{region '#Template'}
	{attribute 'Version' := '1.2.0.0'}
	{attribute 'Tags' := '"LCID": "1031", "Text": "Plant, Weatherstation, Draft"'}
	{attribute 'Tags' := '"LCID": "1033", "Text": "Plant, Weatherstation, Draft"'}
	{attribute 'Description' := '"LCID": "1031", "Text": "Vorlage-Template: beinhaltet alle Objekte, die Eingangsverknüpfung zu diesen muss vom Anwender erstellt werden"'}
	{attribute 'Description' := '"LCID": "1033", "Text": "Draft-template: contains all objects to be connected to appropriate inputs by the user"'}
{endregion}
FUNCTION_BLOCK FB_BA_WeatherStation_Draft EXTENDS FB_BA_View
VAR_INPUT CONSTANT
	Dstb						: FB_BA_SensorBinary;
	Rain						: FB_BA_SensorBinary;
	WthT						: FB_BA_SensorAnalog;
	DewPtT						: FB_BA_SensorAnalog; 
	PrssAbs						: FB_BA_SensorAnalog;
	PrssRel						: FB_BA_SensorAnalog;
	HumAbs						: FB_BA_SensorAnalog;
	HumRel						: FB_BA_SensorAnalog;
	Brightness					: FB_BA_MeasuredValueCardinal;
	Dawn						: FB_BA_SensorAnalog;
	GlobRadn					: FB_BA_SensorAnalog;      
	WndDir						: FB_BA_SensorAnalog;
	WndSpd						: FB_BA_SensorAnalog; 
	Latd						: FB_BA_SensorAnalog;  
	Lngt						: FB_BA_SensorAnalog; 
	SunAzm						: FB_BA_SensorAnalog;
	SunElv						: FB_BA_SensorAnalog;                 
END_VAR	

VAR
	WeatherStation				: FB_BA_RawPublisher;
	stWeatherStation			: ST_BA_WeatherStation;
	stDateTime_PLACEHOLDER		: TIMESTRUCT;			// Placeholder-variable, so the template can be compiled correctly
														// to be replaced by an appropriate timestruct
END_VAR

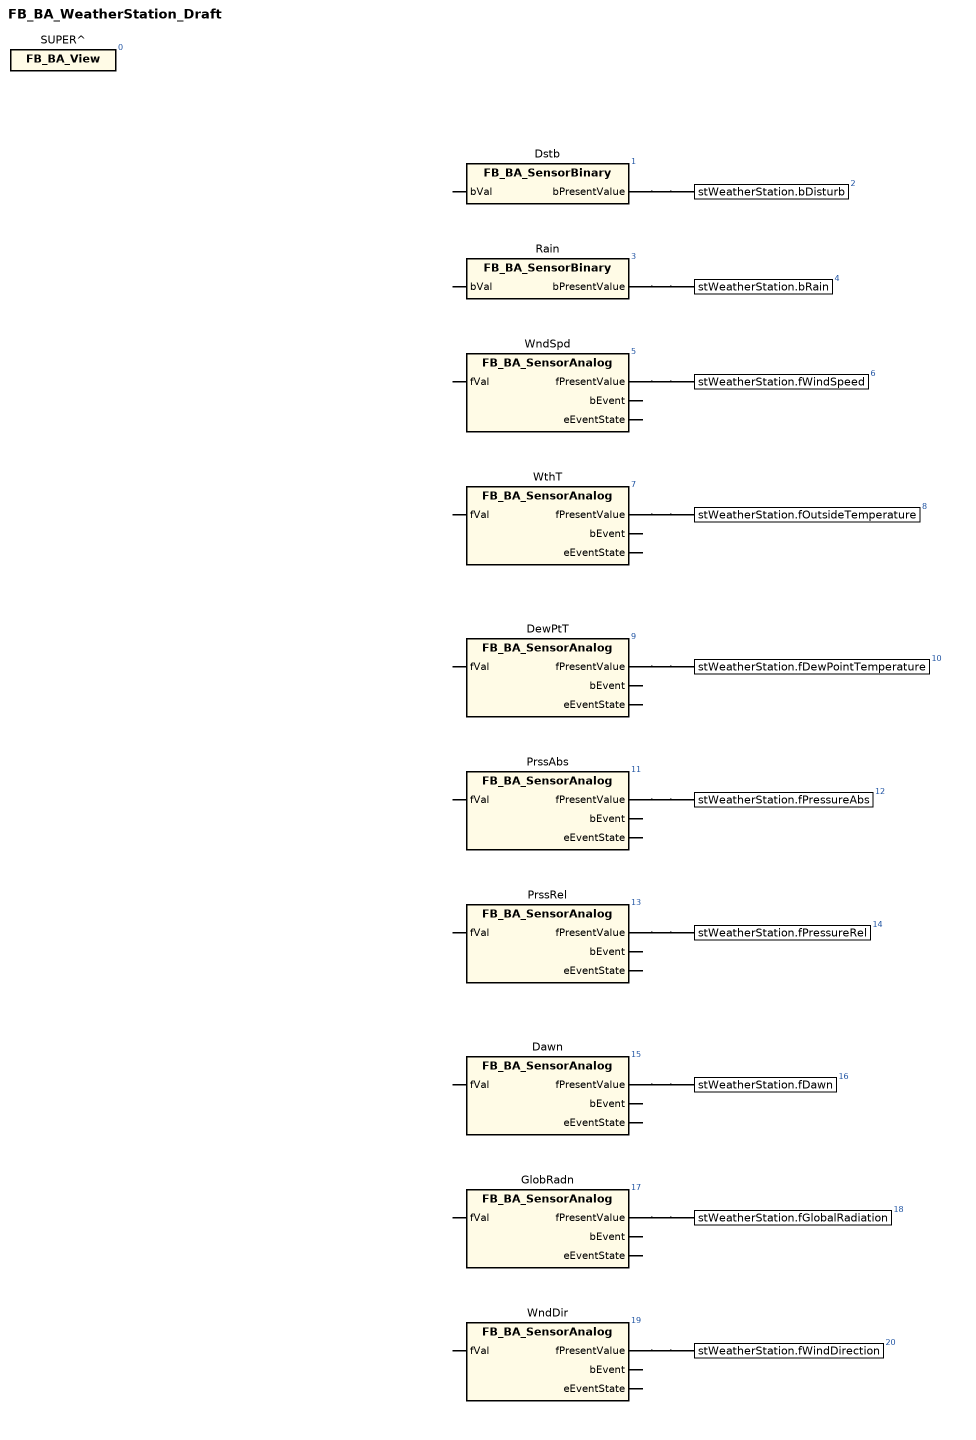
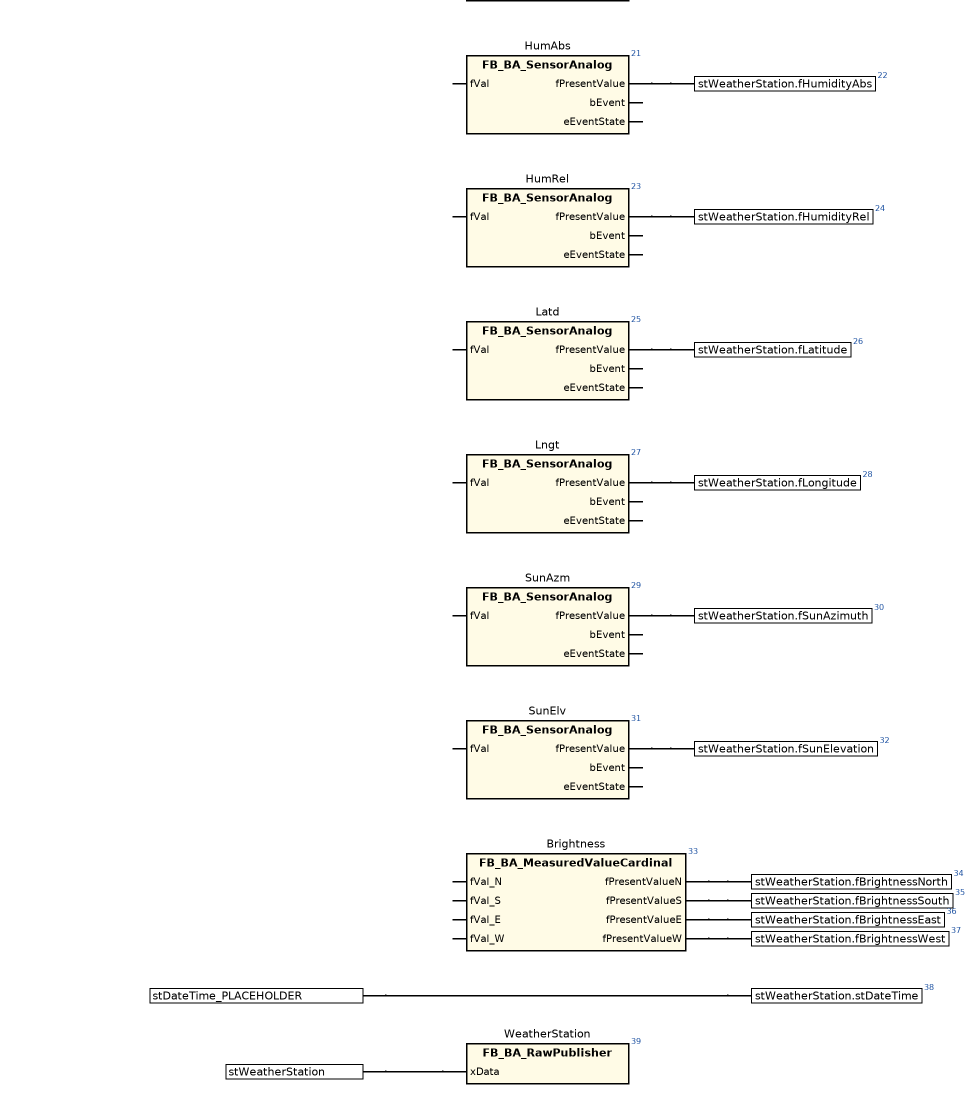
SUPER^(); // FB_BA_View
Dstb(); // FB_BA_SensorBinary
stWeatherStation.bDisturb := Dstb.bPresentValue;
Rain(); // FB_BA_SensorBinary
stWeatherStation.bRain := Rain.bPresentValue;
WndSpd(); // FB_BA_SensorAnalog
stWeatherStation.fWindSpeed := WndSpd.fPresentValue;
WthT(); // FB_BA_SensorAnalog
stWeatherStation.fOutsideTemperature := WthT.fPresentValue;
DewPtT(); // FB_BA_SensorAnalog
stWeatherStation.fDewPointTemperature := DewPtT.fPresentValue;
PrssAbs(); // FB_BA_SensorAnalog
stWeatherStation.fPressureAbs := PrssAbs.fPresentValue;
PrssRel(); // FB_BA_SensorAnalog
stWeatherStation.fPressureRel := PrssRel.fPresentValue;
Dawn(); // FB_BA_SensorAnalog
stWeatherStation.fDawn := Dawn.fPresentValue;
GlobRadn(); // FB_BA_SensorAnalog
stWeatherStation.fGlobalRadiation := GlobRadn.fPresentValue;
WndDir(); // FB_BA_SensorAnalog
stWeatherStation.fWindDirection := WndDir.fPresentValue;
HumAbs(); // FB_BA_SensorAnalog
stWeatherStation.fHumidityAbs := HumAbs.fPresentValue;
HumRel(); // FB_BA_SensorAnalog
stWeatherStation.fHumidityRel := HumRel.fPresentValue;
Latd(); // FB_BA_SensorAnalog
stWeatherStation.fLatitude := Latd.fPresentValue;
Lngt(); // FB_BA_SensorAnalog
stWeatherStation.fLongitude := Lngt.fPresentValue;
SunAzm(); // FB_BA_SensorAnalog
stWeatherStation.fSunAzimuth := SunAzm.fPresentValue;
SunElv(); // FB_BA_SensorAnalog
stWeatherStation.fSunElevation := SunElv.fPresentValue;
Brightness(); // FB_BA_MeasuredValueCardinal
stWeatherStation.fBrightnessNorth := Brightness.fPresentValueN;
stWeatherStation.fBrightnessSouth := Brightness.fPresentValueS;
stWeatherStation.fBrightnessEast := Brightness.fPresentValueE;
stWeatherStation.fBrightnessWest := Brightness.fPresentValueW;
stWeatherStation.stDateTime := stDateTime_PLACEHOLDER;
WeatherStation(xData := stWeatherStation); // FB_BA_RawPublisher

METHOD FB_init : BOOL
VAR_INPUT
	bInitRetains : BOOL; // if TRUE, the retain variables are initialized (warm start / cold start)
	bInCopyCode : BOOL;  // if TRUE, the instance afterwards gets moved into the copy code (online change)
END_VAR
	Dstb.iParent							:= THIS^;
	Dstb.iLabel 							:= LblAggregates_WeatherStation;							
	Dstb.sObjectName						:= '{Idx=01}';
	Dstb.eDPADMode							:= E_BA_DPADMode.eInclude;		
	Dstb.Input.sActiveText 					:= txtEvent_Triggered;       
	Dstb.Input.sInactiveText 				:= txtEvent_Normal;          
	Dstb.Input.nEventClassID				:= EC_ID.NC30;
	Dstb.Input.aEventTransitionText[1]		:= txtEvent_Triggered;       
	Dstb.Input.aEventTransitionText[2]		:= txtEvent_Error;           
	Dstb.Input.aEventTransitionText[3]		:= txtEvent_Normal;          
	Dstb.Input.bEventDetectionEnable		:= TRUE;                     
                        	
	Rain.iParent							:= THIS^;
	Rain.iLabel 							:= LblAggregates_RainSensor;							
	Rain.sObjectName						:= '{Idx=01}';
	Rain.eDPADMode							:= E_BA_DPADMode.eInclude;		
	Rain.Input.iLabel	 					:= LblFunctions_Status;
	Rain.Input.sActiveText 					:= txtEvent_Yes;
	Rain.Input.sInactiveText 				:= txtEvent_No;
	Rain.Input.nEventClassID				:= EC_ID.NC60;
	Rain.Input.aEventTransitionText[1]		:= txtEvent_No;
	Rain.Input.aEventTransitionText[2]		:= txtEvent_None;
	Rain.Input.aEventTransitionText[3]		:= txtEvent_Yes;
	Rain.Input.bEventDetectionEnable		:= FALSE;	
                        	
	WthT.iParent							:= THIS^;
	WthT.iLabel 							:= LblAggregates_TemperatureOutside;
	WthT.sObjectName						:= '{Idx=01}';
	WthT.eDPADMode							:= E_BA_DPADMode.eInclude;
	WthT.MV.eUnit 							:= E_BA_Unit.eTemperature_DegreesCelsius;	
	WthT.MV.eEnPlantLock					:= E_BA_LockPriority.eNoLock;
                    						
	DewPtT.iParent							:= THIS^;
	DewPtT.iLabel 							:= LblAggregates_TemperatureDewPoint;
	DewPtT.sObjectName						:= '{Idx=01}';
	DewPtT.eDPADMode						:= E_BA_DPADMode.eInclude;
	DewPtT.MV.eUnit							:= E_BA_Unit.eTemperature_DegreesCelsius;
	DewPtT.MV.eEnPlantLock					:= E_BA_LockPriority.eNoLock;
                        	
	PrssAbs.iParent							:= THIS^;
	PrssAbs.iLabel 							:= LblAggregates_PressureAbsolute;
	PrssAbs.sObjectName						:= '{Idx=01}';
	PrssAbs.eDPADMode						:= E_BA_DPADMode.eInclude;
	PrssAbs.MV.eUnit						:= E_BA_Unit.ePressure_Hectopascals;
	PrssAbs.MV.eEnPlantLock					:= E_BA_LockPriority.eNoLock;
                        					
	PrssRel.iParent							:= THIS^;
	PrssRel.iLabel 							:= LblAggregates_PressureRelative;
	PrssRel.sObjectName						:= '{Idx=01}';
	PrssRel.eDPADMode						:= E_BA_DPADMode.eInclude;
	PrssRel.MV.eUnit						:= E_BA_Unit.ePressure_Hectopascals;
	PrssRel.MV.eEnPlantLock					:= E_BA_LockPriority.eNoLock;
                        	
	HumAbs.iParent							:= THIS^;
	HumAbs.iLabel 							:= LblAggregates_AbsoluteHumidtiyOutsideAir;
	HumAbs.sObjectName						:= '{Idx=01}';
	HumAbs.eDPADMode						:= E_BA_DPADMode.eInclude;												
	HumAbs.MV.eUnit							:= E_BA_Unit.eHumidity_GramsOfWaterPerKilogramDryAir;
	HumAbs.MV.eEnPlantLock					:= E_BA_LockPriority.eNoLock;
                        					
	HumRel.iParent							:= THIS^;
	HumRel.iLabel 							:= LblAggregates_RelativeHumidityOutsideAir;	
	HumRel.sObjectName						:= '{Idx=01}';
	HumRel.eDPADMode						:= E_BA_DPADMode.eInclude;		
	HumRel.MV.eUnit							:= E_BA_Unit.eHumidity_PercentRelativeHumidity;
	HumRel.MV.eEnPlantLock					:= E_BA_LockPriority.eNoLock;
                        	
	Brightness.iParent						:= THIS^;
	Brightness.iLabel						:= LblAggregates_Brightness;  
	Brightness.MV_N.eUnit					:= E_BA_Unit.eLight_Luxes;
	Brightness.MV_N.sObjectName				:= '{Idx=01}';
	Brightness.MV_N.eEnPlantLock			:= E_BA_LockPriority.eNoLock;
	Brightness.MV_S.eUnit					:= E_BA_Unit.eLight_Luxes;
	Brightness.MV_S.sObjectName				:= '{Idx=02}';
	Brightness.MV_S.eEnPlantLock			:= E_BA_LockPriority.eNoLock;
	Brightness.MV_E.eUnit					:= E_BA_Unit.eLight_Luxes;
	Brightness.MV_E.sObjectName				:= '{Idx=03}';
	Brightness.MV_E.eEnPlantLock			:= E_BA_LockPriority.eNoLock;
	Brightness.MV_W.eUnit					:= E_BA_Unit.eLight_Luxes;
	Brightness.MV_W.sObjectName				:= '{Idx=04}';
	Brightness.MV_W.eEnPlantLock			:= E_BA_LockPriority.eNoLock;

	Dawn.iParent							:= THIS^;
	Dawn.iLabel 							:= LblAggregates_Dawn;
	Dawn.sObjectName						:= '{Idx=01}';
	Dawn.eDPADMode							:= E_BA_DPADMode.eInclude;
	Dawn.MV.eUnit							:= E_BA_Unit.eTemperature_DegreesCelsius;
	Dawn.MV.eEnPlantLock					:= E_BA_LockPriority.eNoLock;
                        	
	GlobRadn.iParent						:= THIS^;
	GlobRadn.iLabel 						:= LblAggregates_SolarRadiation;
	GlobRadn.sObjectName					:= '{Idx=01}';
	GlobRadn.eDPADMode						:= E_BA_DPADMode.eInclude;
	GlobRadn.MV.eUnit						:= E_BA_Unit.eLight_WattsPerSquareMeter;
	GlobRadn.MV.eEnPlantLock				:= E_BA_LockPriority.eNoLock;
                        	
	WndDir.iParent							:= THIS^;
	WndDir.iLabel 							:= LblAggregates_WindDirection;
	WndDir.sObjectName						:= '{Idx=01}';
	WndDir.eDPADMode						:= E_BA_DPADMode.eInclude;
	WndDir.MV.eUnit							:= E_BA_Unit.eOther_DegreesAngular;
	WndDir.MV.eEnPlantLock					:= E_BA_LockPriority.eNoLock;
                        					
	WndSpd.iParent							:= THIS^;
	WndSpd.iLabel 							:= LblAggregates_WindSpeed;		
	WndSpd.sObjectName						:= '{Idx=01}';
	WndSpd.eDPADMode						:= E_BA_DPADMode.eInclude;
	WndSpd.MV.eUnit							:= E_BA_Unit.eVelocity_MetersPerSecond;
	WndSpd.MV.eEnPlantLock					:= E_BA_LockPriority.eNoLock;
                        	
	Latd.iParent							:= THIS^;
	Latd.iLabel 							:= LblAggregates_GeoLatitude;	
	Latd.sObjectName						:= '{Idx=01}';
	Latd.eDPADMode							:= E_BA_DPADMode.eInclude;	
	Latd.MV.eUnit							:= E_BA_Unit.eOther_DegreesAngular;
	Latd.MV.eEnPlantLock					:= E_BA_LockPriority.eNoLock;
                        					
	Lngt.iParent							:= THIS^;
	Lngt.iLabel 							:= LblAggregates_GeoLongitude;
	Lngt.sObjectName						:= '{Idx=01}';
	Lngt.eDPADMode							:= E_BA_DPADMode.eInclude;
	Lngt.MV.eUnit							:= E_BA_Unit.eOther_DegreesAngular;
	Lngt.MV.eEnPlantLock					:= E_BA_LockPriority.eNoLock;
                        	
	SunAzm.iParent							:= THIS^;
	SunAzm.iLabel 							:= LblAggregates_SunAzimuth;	
	SunAzm.sObjectName						:= '{Idx=01}';
	SunAzm.eDPADMode						:= E_BA_DPADMode.eInclude;								
	SunAzm.MV.eUnit							:= E_BA_Unit.eOther_DegreesAngular;
	SunAzm.MV.eEnPlantLock					:= E_BA_LockPriority.eNoLock;
                        	
	SunElv.iParent							:= THIS^;
	SunElv.iLabel 							:= LblAggregates_SunElevation;	
	SunElv.sObjectName						:= '{Idx=01}';
	SunElv.eDPADMode						:= E_BA_DPADMode.eInclude;			
	SunElv.MV.eUnit							:= E_BA_Unit.eOther_DegreesAngular;
	SunElv.MV.eEnPlantLock					:= E_BA_LockPriority.eNoLock;
END_METHOD

END_FUNCTION_BLOCK

(* stored: Version 1.1.0.1, ProductVersion 3.1.4024.9
   POU FB_BA_WeatherStation_Draft: Id {b3a78f62-6f00-4efa-99db-c325823b0792}, SpecialFunc None
   Method FB_init: Id {3b61fef1-ad4e-4ecd-ad06-993193ed1aac} *)
